// Both thresholds use the same engineering unit as the conditioned PV.
// The default equal thresholds are deliberately invalid until configured.
TYPE ST_Hysteresis_Cfg :
STRUCT
    low        : REAL := 0.0;
    high       : REAL := 0.0;
    onBelowLow : BOOL := TRUE; // TRUE for heating/fill, FALSE for cooling/vent.
END_STRUCT
END_TYPE

(* stored: Version 1.1.0.1, ProductVersion 3.1.4026.12
   DUT ST_Hysteresis_Cfg: Id {c7452881-2445-4dc0-9d0a-bb32c542802d} *)
